FUNCTION "Scale_PT100" : Real
{ S7_Optimized_Access := 'TRUE' }
AUTHOR : 'Searinox(Gerrit_Vogtlaender)'
FAMILY : AKK
VERSION : 0.1
   VAR_INPUT
      value : Int;
   END_VAR

   VAR_TEMP
      t_norm : Real;
   END_VAR


BEGIN
	#t_norm := NORM_X(MIN := "AnalogMin", VALUE := #value, MAX := "AnalogMax");
	#Scale_PT100 := LREAL_TO_REAL(SCALE_X(MIN := 0.0, VALUE := #t_norm, MAX := 100.0));
END_FUNCTION

